// TIA Portal V18 export
TYPE "LGasp_typeHMI_ListaProf"
// stored: IsFailsafeCompliant false
   STRUCT
      lista_pezzi : Array[1.."NumMaxPezziProfila"] of "LGasp_typePzoListaProfila";
      nome_articolo_pezzi : Array[1.."NumMaxPezziProfila"] of WString[30];   // il nome dell'articolo viaggia su un array separata perchè tra due plc non si possono passare WSTRING (21010012)
      backup_lista_pezzi : Array[1.."NumMaxPezziProfila"] of "LGasp_typePzoListaProfila";
      pezzo_fatto : "LGasp_typePzoListaProfila";
      abilitata : Bool;
      io_togli_pzo : Bool;
      io_cancella_lista : Bool;
      io_inserisci_pzo_buono : Bool;
      io_inserisci_pzo_scarto : Bool;
      io_recupera_lista { ExternalAccessible := 'False'; ExternalVisible := 'False'; ExternalWritable := 'False'} : Bool;
      listaVuota { ExternalAccessible := 'False'; ExternalVisible := 'False'; ExternalWritable := 'False'} : Bool;
      listaPiena { ExternalAccessible := 'False'; ExternalVisible := 'False'; ExternalWritable := 'False'} : Bool;
   END_STRUCT;
END_TYPE
